FUNCTION_BLOCK FB_TrajMoveJ EXTENDS FB_TrajBase
VAR_OUTPUT
END_VAR
VAR
	// move vector in joint space
	m_moveDir : Vec7d;
	m_moveDistance :LREAL;
	
	// doubleS planning for move distance
	m_doubleS :FB_BasicDoubleS;
END_VAR

METHOD evaluate : BOOL
VAR_INPUT
	t :LREAL;
END_VAR

VAR_IN_OUT
	jntPos,jntVel, jntAcc :vec7d;
END_VAR
VAR
	q,q_dot,q_ddot :LREAL;
END_VAR
evaluate:=m_doubleS.evaluate(t,q=>q,q_dot=>q_dot, q_ddot=>q_dot);
IF evaluate =FALSE THEN
	RETURN;
END_IF

jntPos := multiNumVec7(q, m_moveDir);
jntVel := multiNumVec7(q_dot, m_moveDir);
jntAcc := multiNumVec7(q_ddot, m_moveDir);
END_METHOD

METHOD init : BOOL
VAR_IN_OUT CONSTANT
	i_startJntPos :Vec7d;
	i_targetJntPos :Vec7d;
	i_maxJntVel : Vec7d;
	i_maxJntAcc : Vec7d;
	i_maxJntJerk :Vec7d;
END_VAR
VAR 
	i:INT;
	maxV, maxA, maxJ :LREAL;
	q:ARRAY[1..2] OF LREAL;
	v:ARRAY[1..2] OF LREAL;
END_VAR
m_moveDir:=subVec7(i_targetJntPos, i_startJntPos);
m_moveDistance := normVec7(m_moveDir);

IF(m_moveDistance<g_smallNum) THEN
	m_moveDir:=multiNumVec7(1/7, g_onesVec7d);;
ELSE
	m_moveDir:=multiNumVec7(1/m_moveDistance, m_moveDir);
END_IF

// determian max vel/acc/jerk
maxV:=g_largeNum;
maxA:=g_largeNum;
maxJ:=g_largeNum;
FOR i :=1 TO 7 DO 
	IF ABS(m_moveDir[i])>g_smallNum THEN
		maxV := MIN (maxV, ABS(i_maxJntVel[i]/m_moveDir[i]));
		maxA := MIN (maxA, ABS(i_maxJntAcc[i]/m_moveDir[i]));
		maxJ := MIN (maxJ, ABS(i_maxJntJerk[i]/m_moveDir[i]));
	END_IF
END_FOR

// planning for moving distance
q[1]:=0;
q[2]:=m_moveDistance;
v[1]:=0;
v[2]:=0;
m_doubleS.init(q,v, maxV, maxA, maxJ);
m_duration:=m_doubleS.duration;
m_isGenerated:=m_doubleS.isGene;
END_METHOD

END_FUNCTION_BLOCK

(* stored: Version 1.1.0.1, ProductVersion 3.1.4024.12
   POU FB_TrajMoveJ: Id {02514d4f-2747-4c08-923c-ad3b27b8c50b}, SpecialFunc None
   Method evaluate: Id {87b67f15-ec4f-4ac3-937c-bcf7ce0e7ad6}
   Method init: Id {c13d028d-f18d-482b-a054-8ada64dcb420} *)
